// TIA Portal V19 export
DATA_BLOCK "InstLAF_Checksum"   // DB121
AUTHOR : Siemens Digital Industries
FAMILY : LAF
VERSION : 1.2
// stored: AssignedProDiagFB ProDiag, InstanceOfName LAF_Checksum, InstanceOfType FB
"LAF_Checksum"
   // VAR_INPUT
   //    plantIdentifier { ExternalAccessible := 'False'; ExternalVisible := 'False'; ExternalWritable := 'False'} : WString[24];
   //    textListId { ExternalAccessible := 'False'; ExternalVisible := 'False'; ExternalWritable := 'False'} : Int;
   //    dateTime { ExternalAccessible := 'False'; ExternalVisible := 'False'; ExternalWritable := 'False'} : Date_And_Time;
   //    readChecksum { ExternalAccessible := 'False'; ExternalVisible := 'False'; ExternalWritable := 'False'} : Bool;
   //    ack { ExternalAccessible := 'False'; ExternalVisible := 'False'; ExternalWritable := 'False'} : Bool;
   //    hideMessageStandard { ExternalAccessible := 'False'; ExternalVisible := 'False'; ExternalWritable := 'False'} : Bool;
   //    hideMessageSafety { ExternalAccessible := 'False'; ExternalVisible := 'False'; ExternalWritable := 'False'} : Bool;
   //    hideMessageTextlist { ExternalAccessible := 'False'; ExternalVisible := 'False'; ExternalWritable := 'False'} : Bool;
   // END_VAR
   // VAR_OUTPUT
   //    generalMessage { ExternalAccessible := 'False'; ExternalVisible := 'False'; ExternalWritable := 'False'} : Bool;
   // END_VAR
   // VAR_IN_OUT
   //    checksumHmi : "LAF_typeChecksum";
   // END_VAR
   // VAR
   //    statReadChecksumStorage { ExternalAccessible := 'False'; ExternalVisible := 'False'; ExternalWritable := 'False'} : Bool;
   //    statChecksumStandard { ExternalAccessible := 'False'; ExternalVisible := 'False'; ExternalWritable := 'False'} : Array[0..7] of Byte;
   //    statChecksumStafety { ExternalAccessible := 'False'; ExternalVisible := 'False'; ExternalWritable := 'False'} : Array[0..7] of Byte;
   //    statChecksumTextlists { ExternalAccessible := 'False'; ExternalVisible := 'False'; ExternalWritable := 'False'} : Array[0..7] of Byte;
   //    statChecksumStandOldNull { ExternalAccessible := 'False'; ExternalVisible := 'False'; ExternalWritable := 'False'} : Bool;
   //    statChecksumSafeOldNull { ExternalAccessible := 'False'; ExternalVisible := 'False'; ExternalWritable := 'False'} : Bool;
   //    statChecksumTextlOldNull { ExternalAccessible := 'False'; ExternalVisible := 'False'; ExternalWritable := 'False'} : Bool;
   //    statChecksumStandDiff { ExternalAccessible := 'False'; ExternalVisible := 'False'; ExternalWritable := 'False'} : Bool;
   //    statChecksumSafeDiff { ExternalAccessible := 'False'; ExternalVisible := 'False'; ExternalWritable := 'False'} : Bool;
   //    statChecksumTextlDiff { ExternalAccessible := 'False'; ExternalVisible := 'False'; ExternalWritable := 'False'} : Bool;
   //    instGetChecksum1 { ExternalAccessible := 'False'; ExternalVisible := 'False'; ExternalWritable := 'False'} : GetChecksum;
   //    instGetChecksum2 { ExternalAccessible := 'False'; ExternalVisible := 'False'; ExternalWritable := 'False'} : GetChecksum;
   //    instGetChecksum3 { ExternalAccessible := 'False'; ExternalVisible := 'False'; ExternalWritable := 'False'} : GetChecksum;
   //    statRetValHta { ExternalAccessible := 'False'; ExternalVisible := 'False'; ExternalWritable := 'False'} : "LAF_typeChecksumCatWord";
   //    statRisEdgeDiff { ExternalAccessible := 'False'; ExternalVisible := 'False'; ExternalWritable := 'False'} : "LAF_typeChecksumCatBool";
   //    statMessageStandModified { ExternalAccessible := 'False'; ExternalVisible := 'False'; ExternalWritable := 'False'} : Bool;
   //    statMessageSafeModified { ExternalAccessible := 'False'; ExternalVisible := 'False'; ExternalWritable := 'False'} : Bool;
   //    statMessageTextlModified { ExternalAccessible := 'False'; ExternalVisible := 'False'; ExternalWritable := 'False'} : Bool;
   //    statWarnNoStandard { ExternalAccessible := 'False'; ExternalVisible := 'False'; ExternalWritable := 'False'} : UInt;
   //    statWarnNoSafety { ExternalAccessible := 'False'; ExternalVisible := 'False'; ExternalWritable := 'False'} : UInt;
   //    statWarnNoTextlist { ExternalAccessible := 'False'; ExternalVisible := 'False'; ExternalWritable := 'False'} : UInt;
   // END_VAR
BEGIN
END_DATA_BLOCK
